// TIA Portal V16 export
// export: Created 2021-11-12T13:31:44.2909433Z, ExportSetting WithDefaults, DisplayName Totally Integrated Automation Portal, DisplayVersion V16 Update 3, DisplayName TIA Portal Version Control Interface, DisplayVersion V16 Update 2, DisplayName TIA Portal Openness, DisplayVersion V16 Update 3, DisplayName SINAMICS Startdrive Advanced, DisplayVersion V16 Update 5, DisplayName SINAMICS Startdrive G130, G150, S120, S150, SINAMICS MV, S210, DisplayVersion V16 Update 5, DisplayName SINAMICS Startdrive G110M, G120, G120C, G120D, G120P, G115D, DisplayVersion V16 Update 5, DisplayName STEP 7 Professional, DisplayVersion V16 Update 3, DisplayName STEP 7 Safety, DisplayVersion V16, DisplayName WinCC UA Professional, DisplayVersion V16 Update 3
FUNCTION_BLOCK "STD_Siemens_MC_Encoder"   // FB31, LAD
TITLE = Siemens MC-Encoder Multiturn 27-bit
{ S7_Optimized_Access := 'TRUE' }
VERSION : 0.1
// MICE standard block 
// Communication with Siemens MC-Encoder Multiturn 27-bit (6FX2001-5FN25)
// 
// 
// Version              Created                        by             Comment
// 0.1                      16.7.2019                   JKu          initial version
// stored: AutoNumber true, IsIECCheckEnabled false, IsRetainMemResEnabled false, MemoryReserve 100, SetENOAutomatically false, UDAEnableTagReadback false
   VAR_INPUT
      IW_HWID : HW_SUBMODULE;
      IB1Preset : Bool;   // Set previously configured home position (absolute)
      IB1Ack : Bool;   // Alarm reset
      IB1AlarmSuppress : Bool;   // Alarm suppression
   END_VAR
   VAR_OUTPUT
      OS_Status : Struct
         Main : "UDT_Status_main";
         Specific : "UDT_MCEncoder_Status_specific";
         Error : "UDT_Error01";
      END_STRUCT;
      OR_AbsPosUnits : Real;   // Absolute actual position [mm]
   END_VAR
   VAR_IN_OUT
      XS_Parameter : "UDT_MCEnkoder_Parameter";   // Individual parameter structure
      XS_Command : "UDT_MCEnkoder_Command";
   END_VAR
   VAR
      SS_Alarm : Struct   // Device alarms
         SensorError : Bool;   // Error in the processing of the sensor signal
         CommandNotSupported : Bool;   // Optional command (in G1_STW) not supported.
         PLCSignOfLifeFailure : Bool;   // The number of permissible failures of the masters
         SynchronizationFault : Bool;   // The number of permissible failures for the bus cycle
         Overflow : Bool;   // The position value in G1_XIST1 overflow
         InvalidData : Bool;   // Data from encoder is invalid and encoder does not respond to commands
         res0_6 : Bool;
         res0_7 : Bool;
      END_STRUCT;
      SS_Warning : Struct   // Device warnings
         res0_0 : Bool;
         res0_1 : Bool;
         res0_2 : Bool;
         res0_3 : Bool;
         res0_4 : Bool;
         res0_5 : Bool;
         res0_6 : Bool;
         res0_7 : Bool;
      END_STRUCT;
   END_VAR
   VAR_TEMP
      TS_Parameter : "UDT_MCEnkoder_Parameter";
      TS_Status : Struct
         Main : "UDT_Status_main";
         Specific : "UDT_MCEncoder_Status_specific";
         Error : "UDT_Error01";
      END_STRUCT;
      TS_InData : "UDT_MCEncoder_I_81";
      TS_OutData : "UDT_MCEncoder_O_81";
      TI_RetVal : Int;
      TI_AbsPosVal : Int;   // Absolute actual position value within one turn
      TR_AbsPosUnits : Real;   // Absolute actual position [mm]
      TI_NoOfRevolution : Int;   // Number of revolutions
      TDWMaskedVal : DWord;   // G1_XIST value masked
      TI_ErrorCode : Int;
      TB1DataValid : Bool;   // Data in G1_XIST1 and G1_ZSW is valid
      TB1 : Bool;
   END_VAR
   VAR CONSTANT
      CI_PulsePerTurn : Int := 8192;   // Resolution
      CI_MaxRevolutions : Int := 16384;   // Maximum number of revolution what the encoder is capable to count
      CI_AbsPosNrOfBits : Int := 13;   // Bit lenght of absolute position value
      CDWMaskAbsPos : DWord := 16#00001FFF;   // Absolute position value mask G1_XIST1
      CDWMaskMultiturnData : DWord := 16#07FFE000;   // Multiturn data mask G1_XIST1
      CDWMaskErrorCode : DWord := 16#00000FFF;   // Error code mask G1_XIST1
   END_VAR
BEGIN

REGION Network 1: Clear temporary variables
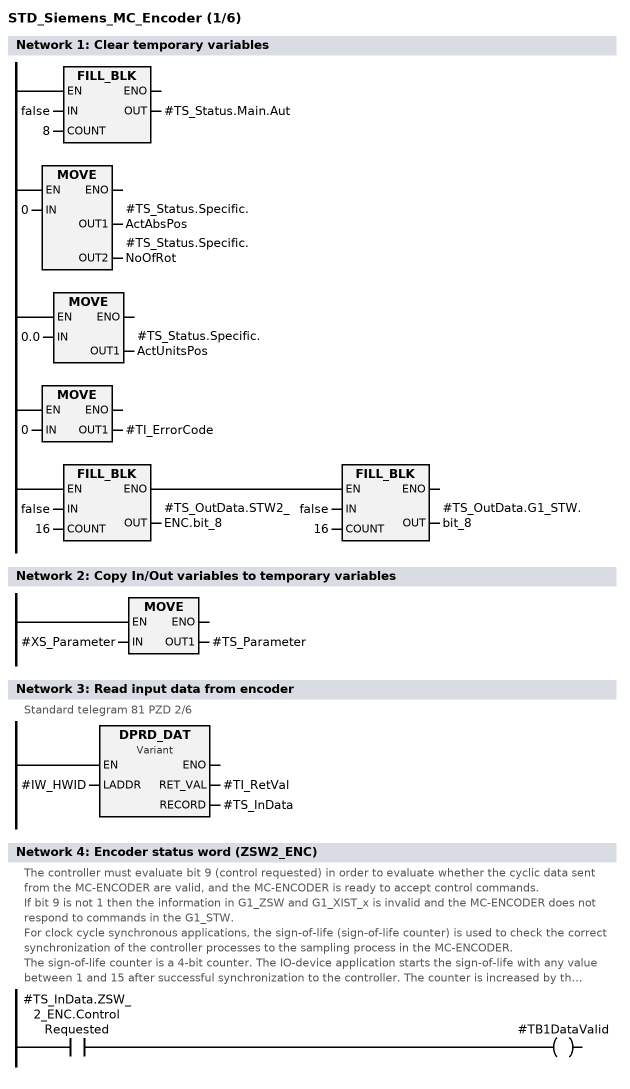
   RUNG wire#powerrail
      FillBlockI(in := false, count := 8, out => #TS_Status.Main.Aut)
   END_RUNG
   RUNG wire#powerrail
      Move(in := 0, out1 => #TS_Status.Specific.ActAbsPos, out2 => #TS_Status.Specific.NoOfRot)
   END_RUNG
   RUNG wire#powerrail
      Move(in := 0.0, out1 => #TS_Status.Specific.ActUnitsPos)
   END_RUNG
   RUNG wire#powerrail
      Move(in := 0, out1 => #TI_ErrorCode)
   END_RUNG
   RUNG wire#powerrail
      FillBlockI(in := false, count := 16, out => #TS_OutData.STW2_ENC.bit_8)
      FillBlockI(in := false, count := 16, out => #TS_OutData.G1_STW.bit_8)
   END_RUNG
   // the same network as SCL:
   FILL_BLK(IN := false, COUNT := 8, OUT => #TS_Status.Main.Aut);
   #TS_Status.Specific.ActAbsPos := 0;
   #TS_Status.Specific.NoOfRot := 0;
   #TS_Status.Specific.ActUnitsPos := 0.0;
   #TI_ErrorCode := 0;
   FILL_BLK(IN := false, COUNT := 16, OUT => #TS_OutData.STW2_ENC.bit_8);
   FILL_BLK(IN := false, COUNT := 16, OUT => #TS_OutData.G1_STW.bit_8);
END_REGION

REGION Network 2: Copy In/Out variables to temporary variables
   RUNG wire#powerrail
      { S7_GenerateENO := "TRUE" } Move(in := #XS_Parameter, out1 => #TS_Parameter)
   END_RUNG
   // the same network as SCL:
   #TS_Parameter := #XS_Parameter;
END_REGION

REGION Network 3: Read input data from encoder
   // Standard telegram 81 PZD 2/6
   RUNG wire#powerrail
      { S7_Templates := "[ptr_type := Variant, laddr_type := HW_IO]" } DPRD_DAT(LADDR := #IW_HWID, RET_VAL => #TI_RetVal, RECORD => #TS_InData)
   END_RUNG
   // the same network as SCL:
   #TI_RetVal := DPRD_DAT(LADDR := #IW_HWID, RECORD => #TS_InData);
END_REGION

REGION Network 4: Encoder status word (ZSW2_ENC)
   // The controller must evaluate bit 9 (control requested) in order to evaluate whether the cyclic data sent from the MC-ENCODER are valid, and the MC-ENCODER is ready to accept control commands.
   // If bit 9 is not 1 then the information in G1_ZSW and G1_XIST_x is invalid and the MC-ENCODER does not respond to commands in the G1_STW.
   // 
   // For clock cycle synchronous applications, the sign-of-life (sign-of-life counter) is used to check the correct synchronization of the controller processes to the sampling process in the MC-ENCODER.
   // The sign-of-life counter is a 4-bit counter. The IO-device application starts the sign-of-life with any value between 1 and 15 after successful synchronization to the controller. The counter is increased by the IO-device in every data cycle. Valid values for the IO-device sign-of-life are 1 to 15, "0" indicates an error and is left out in normal operation.
   // 
   // If the MC-ENCODER identifies an error in the controller sign-of-life, then it stops sending the sign-of-life to the controller. This means that a missing sign-of-life (=0) from the MC-ENCODER to the controller can also be the consequence of an error in the controller sign-of-life to MCENCODER.
   RUNG wire#powerrail
      Contact( #TS_InData.ZSW_2_ENC.ControlRequested )
      Coil( #TB1DataValid )
   END_RUNG
   // the same network as SCL:
   #TB1DataValid := #TS_InData.ZSW_2_ENC.ControlRequested;
END_REGION

REGION Network 5: Sensor status word (G1_ZSW)
   // Signal G1_ZSW is used to control the state machine of the PROFIdrive encoder channel and is the counterpart to control word G1_STW.
   // 
   // bit 11 - Acknowledgement sensor error in process - Is set while requested error acknowledge is processed. Handshake signal related to G1_STW bit 15.
   // bit 12 - Set preset / shift reference point executed - Acknowledgement for "set preset / request shift".
   // bit 13 - Transmit absolute value cyclically - Acknowledgement for "request absolute value cyclically".
   // bit 14 - Parking sensor activated - Acknowledgement for "activate parking sensor". The encoder transmits no valid position value, sensor errors are reset.
   // bit 15 - Sensor error - Indicates a sensor error. A device specific error code is transmitted in G1_XIST2.
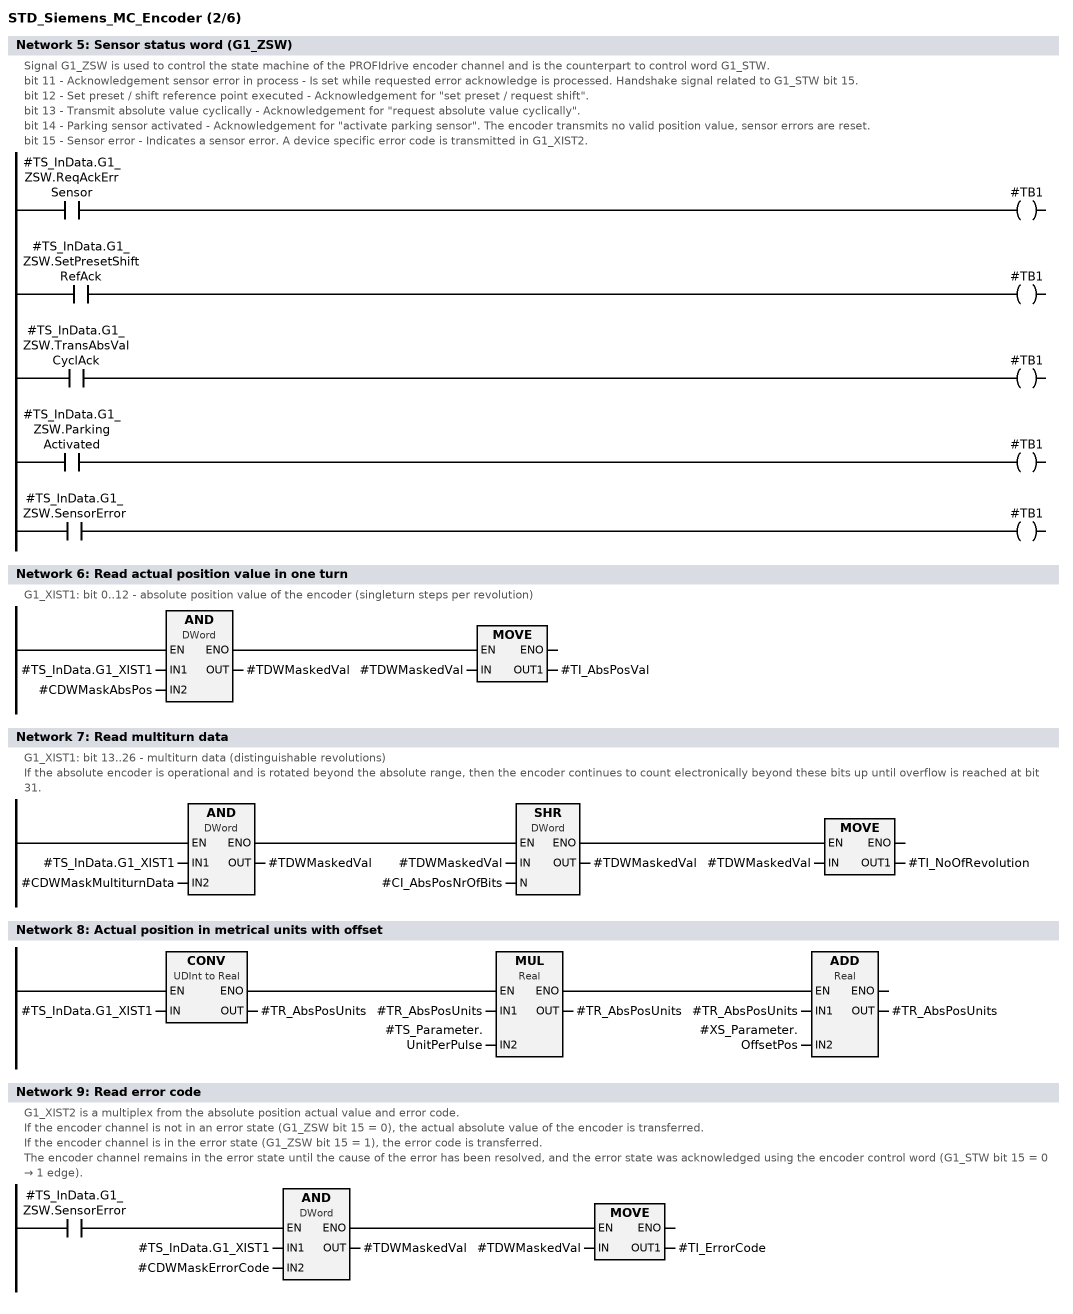
   RUNG wire#powerrail
      Contact( #TS_InData.G1_ZSW.ReqAckErrSensor )
      Coil( #TB1 )
   END_RUNG
   RUNG wire#powerrail
      Contact( #TS_InData.G1_ZSW.SetPresetShiftRefAck )
      Coil( #TB1 )
   END_RUNG
   RUNG wire#powerrail
      Contact( #TS_InData.G1_ZSW.TransAbsValCyclAck )
      Coil( #TB1 )
   END_RUNG
   RUNG wire#powerrail
      Contact( #TS_InData.G1_ZSW.ParkingActivated )
      Coil( #TB1 )
   END_RUNG
   RUNG wire#powerrail
      Contact( #TS_InData.G1_ZSW.SensorError )
      Coil( #TB1 )
   END_RUNG
   // the same network as SCL:
   #TB1 := #TS_InData.G1_ZSW.ReqAckErrSensor;
   #TB1 := #TS_InData.G1_ZSW.SetPresetShiftRefAck;
   #TB1 := #TS_InData.G1_ZSW.TransAbsValCyclAck;
   #TB1 := #TS_InData.G1_ZSW.ParkingActivated;
   #TB1 := #TS_InData.G1_ZSW.SensorError;
END_REGION

REGION Network 6: Read actual position value in one turn
   // G1_XIST1: bit 0..12 - absolute position value of the encoder (singleturn steps per revolution)
   RUNG wire#powerrail
      { S7_Templates := "SrcType := DWord" } And(in1 := #TS_InData.G1_XIST1, in2 := #CDWMaskAbsPos, out => #TDWMaskedVal)
      Move(in := #TDWMaskedVal, out1 => #TI_AbsPosVal)
   END_RUNG
   // the same network as SCL:
   #TDWMaskedVal := #TS_InData.G1_XIST1 AND #CDWMaskAbsPos;
   #TI_AbsPosVal := #TDWMaskedVal;
END_REGION

REGION Network 7: Read multiturn data
   // G1_XIST1: bit 13..26 - multiturn data (distinguishable revolutions)
   // If the absolute encoder is operational and is rotated beyond the absolute range, then the encoder continues to count electronically beyond these bits up until overflow is reached at bit 31.
   RUNG wire#powerrail
      { S7_Templates := "SrcType := DWord" } And(in1 := #TS_InData.G1_XIST1, in2 := #CDWMaskMultiturnData, out => #TDWMaskedVal)
      { S7_Templates := "SrcType := DWord" } Shr(in := #TDWMaskedVal, n := #CI_AbsPosNrOfBits, out => #TDWMaskedVal)
      Move(in := #TDWMaskedVal, out1 => #TI_NoOfRevolution)
   END_RUNG
   // the same network as SCL:
   #TDWMaskedVal := #TS_InData.G1_XIST1 AND #CDWMaskMultiturnData;
   #TDWMaskedVal := SHR(IN := #TDWMaskedVal, N := #CI_AbsPosNrOfBits);
   #TI_NoOfRevolution := #TDWMaskedVal;
END_REGION

REGION Network 8: Actual position in metrical units with offset
   RUNG wire#powerrail
      { S7_Templates := "[SrcType := UDInt, DestType := Real]" } Convert(in := #TS_InData.G1_XIST1, out => #TR_AbsPosUnits)
      { S7_Templates := "SrcType := Real" } Mul(in1 := #TR_AbsPosUnits, in2 := #TS_Parameter.UnitPerPulse, out => #TR_AbsPosUnits)
      { S7_Templates := "SrcType := Real" } Add(in1 := #TR_AbsPosUnits, in2 := #XS_Parameter.OffsetPos, out => #TR_AbsPosUnits)
   END_RUNG
   // the same network as SCL:
   #TR_AbsPosUnits := UDINT_TO_REAL(#TS_InData.G1_XIST1);
   #TR_AbsPosUnits := #TR_AbsPosUnits * #TS_Parameter.UnitPerPulse;
   #TR_AbsPosUnits := #TR_AbsPosUnits + #XS_Parameter.OffsetPos;
END_REGION

REGION Network 9: Read error code
   // G1_XIST2 is a multiplex from the absolute position actual value and error code. 
   // If the encoder channel is not in an error state (G1_ZSW bit 15 = 0), the actual absolute value of the encoder is transferred.
   // If the encoder channel is in the error state (G1_ZSW bit 15 = 1), the error code is transferred.
   // The encoder channel remains in the error state until the cause of the error has been resolved, and the error state was acknowledged using the encoder control word (G1_STW bit 15 = 0 → 1 edge).
   RUNG wire#powerrail
      Contact( #TS_InData.G1_ZSW.SensorError )
      { S7_Templates := "SrcType := DWord" } And(in1 := #TS_InData.G1_XIST1, in2 := #CDWMaskErrorCode, out => #TDWMaskedVal)
      Move(in := #TDWMaskedVal, out1 => #TI_ErrorCode)
   END_RUNG
   // the same network as SCL:
   IF #TS_InData.G1_ZSW.SensorError THEN
       #TDWMaskedVal := #TS_InData.G1_XIST1 AND #CDWMaskErrorCode;
       #TI_ErrorCode := #TDWMaskedVal;
   END_IF;
END_REGION

REGION Network 10: Error evaluation
   // 0x001  Sensor group error - Error in the processing of the sensor signal which causes an invalid Gx_XIST (e.g. electronic malfunction or invalid sensor signal).
   // 0xF01  Command not supported - Optional command (in G1_STW) not supported.
   // 0xF02  Controller sign-of-life failure - The number of permissible failures of the masters sign-of-life was exceeded.
   // 0xF04  Synchronization fault - The number of permissible failures for the bus cycle sign signal was exceeded.
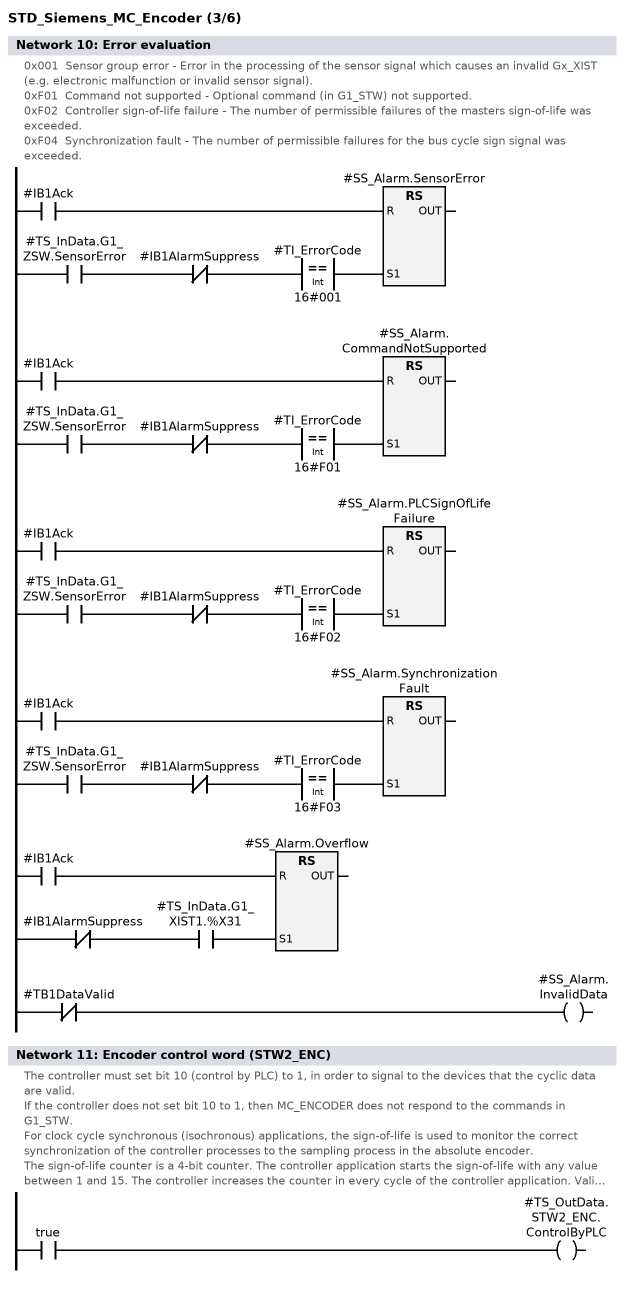
   RUNG wire#powerrail
      Contact( #IB1Ack )
      S_RS(operand := #SS_Alarm.SensorError, s1 := wire#w1)
   END_RUNG
   RUNG wire#powerrail
      Contact( #TS_InData.G1_ZSW.SensorError )
      I_Contact( #IB1AlarmSuppress )
      { S7_Templates := "SrcType := Int" } EQ_Contact(in1 := #TI_ErrorCode, in2 := 16#001)
   END_RUNG wire#w1
   RUNG wire#powerrail
      Contact( #IB1Ack )
      S_RS(operand := #SS_Alarm.CommandNotSupported, s1 := wire#w2)
   END_RUNG
   RUNG wire#powerrail
      Contact( #TS_InData.G1_ZSW.SensorError )
      I_Contact( #IB1AlarmSuppress )
      { S7_Templates := "SrcType := Int" } EQ_Contact(in1 := #TI_ErrorCode, in2 := 16#F01)
   END_RUNG wire#w2
   RUNG wire#powerrail
      Contact( #IB1Ack )
      S_RS(operand := #SS_Alarm.PLCSignOfLifeFailure, s1 := wire#w3)
   END_RUNG
   RUNG wire#powerrail
      Contact( #TS_InData.G1_ZSW.SensorError )
      I_Contact( #IB1AlarmSuppress )
      { S7_Templates := "SrcType := Int" } EQ_Contact(in1 := #TI_ErrorCode, in2 := 16#F02)
   END_RUNG wire#w3
   RUNG wire#powerrail
      Contact( #IB1Ack )
      S_RS(operand := #SS_Alarm.SynchronizationFault, s1 := wire#w4)
   END_RUNG
   RUNG wire#powerrail
      Contact( #TS_InData.G1_ZSW.SensorError )
      I_Contact( #IB1AlarmSuppress )
      { S7_Templates := "SrcType := Int" } EQ_Contact(in1 := #TI_ErrorCode, in2 := 16#F03)
   END_RUNG wire#w4
   RUNG wire#powerrail
      Contact( #IB1Ack )
      S_RS(operand := #SS_Alarm.Overflow, s1 := wire#w5)
   END_RUNG
   RUNG wire#powerrail
      I_Contact( #IB1AlarmSuppress )
      Contact( #TS_InData.G1_XIST1.%X31 )
   END_RUNG wire#w5
   RUNG wire#powerrail
      I_Contact( #TB1DataValid )
      Coil( #SS_Alarm.InvalidData )
   END_RUNG
   // the same network as SCL:
   IF #IB1Ack THEN
       #SS_Alarm.SensorError := FALSE;   // RS flip-flop
   END_IF;
   IF #TS_InData.G1_ZSW.SensorError AND NOT #IB1AlarmSuppress AND (#TI_ErrorCode = 16#001) THEN
       #SS_Alarm.SensorError := TRUE;
   END_IF;
   IF #IB1Ack THEN
       #SS_Alarm.CommandNotSupported := FALSE;   // RS flip-flop
   END_IF;
   IF #TS_InData.G1_ZSW.SensorError AND NOT #IB1AlarmSuppress AND (#TI_ErrorCode = 16#F01) THEN
       #SS_Alarm.CommandNotSupported := TRUE;
   END_IF;
   IF #IB1Ack THEN
       #SS_Alarm.PLCSignOfLifeFailure := FALSE;   // RS flip-flop
   END_IF;
   IF #TS_InData.G1_ZSW.SensorError AND NOT #IB1AlarmSuppress AND (#TI_ErrorCode = 16#F02) THEN
       #SS_Alarm.PLCSignOfLifeFailure := TRUE;
   END_IF;
   IF #IB1Ack THEN
       #SS_Alarm.SynchronizationFault := FALSE;   // RS flip-flop
   END_IF;
   IF #TS_InData.G1_ZSW.SensorError AND NOT #IB1AlarmSuppress AND (#TI_ErrorCode = 16#F03) THEN
       #SS_Alarm.SynchronizationFault := TRUE;
   END_IF;
   IF #IB1Ack THEN
       #SS_Alarm.Overflow := FALSE;   // RS flip-flop
   END_IF;
   IF NOT #IB1AlarmSuppress AND #TS_InData.G1_XIST1.%X31 THEN #SS_Alarm.Overflow := TRUE; END_IF;
   #SS_Alarm.InvalidData := NOT #TB1DataValid;
END_REGION

REGION Network 11: Encoder control word (STW2_ENC)
   // The controller must set bit 10 (control by PLC) to 1, in order to signal to the devices that the cyclic data are valid.
   // If the controller does not set bit 10 to 1, then MC_ENCODER does not respond to the commands in G1_STW.
   // 
   // For clock cycle synchronous (isochronous) applications, the sign-of-life is used to monitor the correct synchronization of the controller processes to the sampling process in the absolute encoder.
   // The sign-of-life counter is a 4-bit counter. The controller application starts the sign-of-life with any value between 1 and 15. The controller increases the counter in every cycle of the controller application. Valid values for the controller sign-of-life are 1 to 15, "0" indicates an error and is left out in normal operation.
   RUNG wire#powerrail
      Contact( true )
      Coil( #TS_OutData.STW2_ENC.ControlByPLC )
   END_RUNG
   // the same network as SCL:
   #TS_OutData.STW2_ENC.ControlByPLC := true;
END_REGION

REGION Network 12: Sensor control word (G1_STW)
   // Signal G1_STW is used to control the state machine of the PROFIdrive encoder channel.
   // 
   // bit 11 - Home position mode - Specifies if the position value shall be set to a previously configured absolute value or shifted by this value. 
   //   0: set home position / preset (absolute) 
   //   1: shift home position / preset (relative = offset)
   // 
   // bit 12 - Set preset / request shift - Preset (resp. shift) is set when changing this bit to "1" (rising edge). Default preset value (shift): 0
   // Note: It can also be parameterized that with a rising edge, the value XIST1 also makes a step.
   // 
   // bit 13 - Request absolute value cyclically - Request of additional cyclic transmission of the absolute actual position in G1_XIST2. If no other data needs to be transferred due to commands or errors the absolute position value will be transmitted automatically.
   // 
   // bit 14 - Activate parking sensor - The encoder is switched inactive and error will be reset. While the encoder is in the parking state, no errors will be generated.
   // 
   // bit 15 - Acknowledging a sensor error - Request to acknowledge / reset a sensor error.
   // 
   // By appropriately parameterizing the absolute encoder, when accepting the preset value, you can set whether this is also directly accepted in G1_XIST1 or G1_XIST3. When the preset value is accepted, this value is also retentively saved automatically. This is to ensure that an absolute value set using preset is also kept after a reset/power up of the encoder.
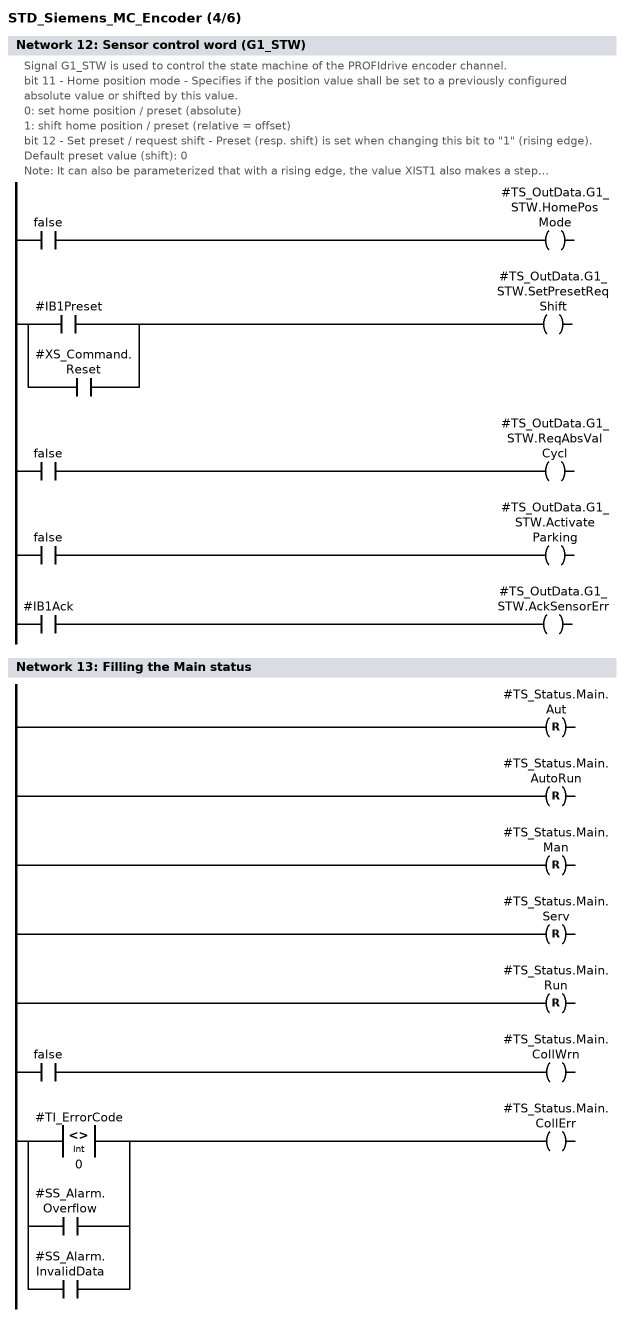
   RUNG wire#powerrail
      Contact( false )
      Coil( #TS_OutData.G1_STW.HomePosMode )
   END_RUNG
   RUNG wire#powerrail
      Contact( #IB1Preset )
      wire#w1
      Coil( #TS_OutData.G1_STW.SetPresetReqShift )
   END_RUNG
   RUNG wire#powerrail
      Contact( #XS_Command.Reset )
   END_RUNG wire#w1
   RUNG wire#powerrail
      Contact( false )
      Coil( #TS_OutData.G1_STW.ReqAbsValCycl )
   END_RUNG
   RUNG wire#powerrail
      Contact( false )
      Coil( #TS_OutData.G1_STW.ActivateParking )
   END_RUNG
   RUNG wire#powerrail
      Contact( #IB1Ack )
      Coil( #TS_OutData.G1_STW.AckSensorErr )
   END_RUNG
   // the same network as SCL:
   #TS_OutData.G1_STW.HomePosMode := false;
   #TS_OutData.G1_STW.SetPresetReqShift := #IB1Preset OR #XS_Command.Reset;
   #TS_OutData.G1_STW.ReqAbsValCycl := false;
   #TS_OutData.G1_STW.ActivateParking := false;
   #TS_OutData.G1_STW.AckSensorErr := #IB1Ack;
END_REGION

REGION Network 13: Filling the Main status
   RUNG wire#powerrail
      R_Coil( #TS_Status.Main.Aut )
   END_RUNG
   RUNG wire#powerrail
      R_Coil( #TS_Status.Main.AutoRun )
   END_RUNG
   RUNG wire#powerrail
      R_Coil( #TS_Status.Main.Man )
   END_RUNG
   RUNG wire#powerrail
      R_Coil( #TS_Status.Main.Serv )
   END_RUNG
   RUNG wire#powerrail
      R_Coil( #TS_Status.Main.Run )
   END_RUNG
   RUNG wire#powerrail
      Contact( false )
      Coil( #TS_Status.Main.CollWrn )
   END_RUNG
   RUNG wire#powerrail
      { S7_Templates := "SrcType := Int" } NE_Contact(in1 := #TI_ErrorCode, in2 := 0)
      wire#w1
      Coil( #TS_Status.Main.CollErr )
   END_RUNG
   RUNG wire#powerrail
      Contact( #SS_Alarm.Overflow )
   END_RUNG wire#w1
   RUNG wire#powerrail
      Contact( #SS_Alarm.InvalidData )
   END_RUNG wire#w1
   // the same network as SCL:
   #TS_Status.Main.Aut := FALSE;
   #TS_Status.Main.AutoRun := FALSE;
   #TS_Status.Main.Man := FALSE;
   #TS_Status.Main.Serv := FALSE;
   #TS_Status.Main.Run := FALSE;
   #TS_Status.Main.CollWrn := false;
   #TS_Status.Main.CollErr := (#TI_ErrorCode <> 0) OR #SS_Alarm.Overflow OR #SS_Alarm.InvalidData;
END_REGION

REGION Network 14: Filling the specific status
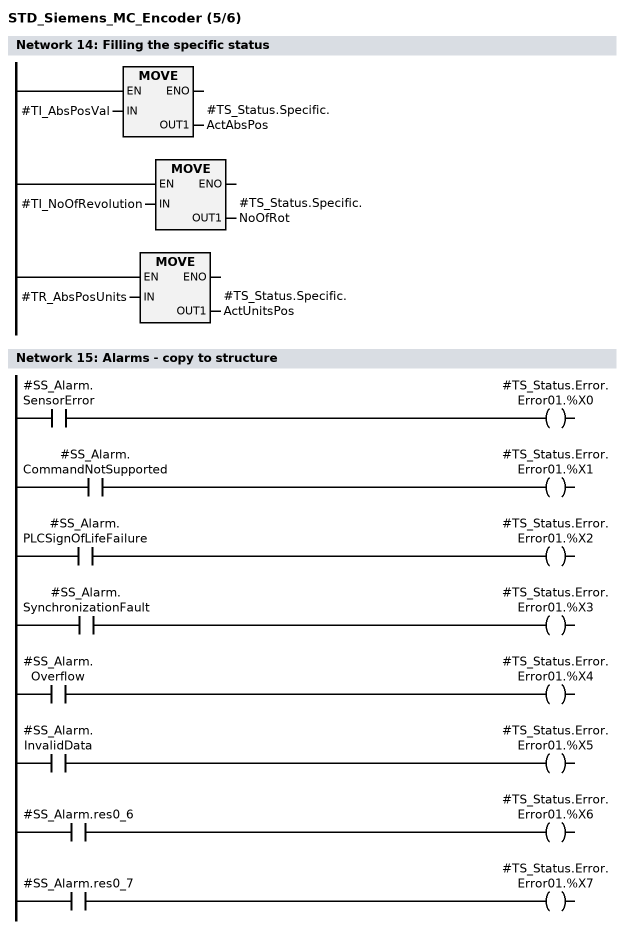
   RUNG wire#powerrail
      Move(in := #TI_AbsPosVal, out1 => #TS_Status.Specific.ActAbsPos)
   END_RUNG
   RUNG wire#powerrail
      Move(in := #TI_NoOfRevolution, out1 => #TS_Status.Specific.NoOfRot)
   END_RUNG
   RUNG wire#powerrail
      Move(in := #TR_AbsPosUnits, out1 => #TS_Status.Specific.ActUnitsPos)
   END_RUNG
   // the same network as SCL:
   #TS_Status.Specific.ActAbsPos := #TI_AbsPosVal;
   #TS_Status.Specific.NoOfRot := #TI_NoOfRevolution;
   #TS_Status.Specific.ActUnitsPos := #TR_AbsPosUnits;
END_REGION

REGION Network 15: Alarms - copy to structure
   RUNG wire#powerrail
      Contact( #SS_Alarm.SensorError )
      Coil( #TS_Status.Error.Error01.%X0 )
   END_RUNG
   RUNG wire#powerrail
      Contact( #SS_Alarm.CommandNotSupported )
      Coil( #TS_Status.Error.Error01.%X1 )
   END_RUNG
   RUNG wire#powerrail
      Contact( #SS_Alarm.PLCSignOfLifeFailure )
      Coil( #TS_Status.Error.Error01.%X2 )
   END_RUNG
   RUNG wire#powerrail
      Contact( #SS_Alarm.SynchronizationFault )
      Coil( #TS_Status.Error.Error01.%X3 )
   END_RUNG
   RUNG wire#powerrail
      Contact( #SS_Alarm.Overflow )
      Coil( #TS_Status.Error.Error01.%X4 )
   END_RUNG
   RUNG wire#powerrail
      Contact( #SS_Alarm.InvalidData )
      Coil( #TS_Status.Error.Error01.%X5 )
   END_RUNG
   RUNG wire#powerrail
      Contact( #SS_Alarm.res0_6 )
      Coil( #TS_Status.Error.Error01.%X6 )
   END_RUNG
   RUNG wire#powerrail
      Contact( #SS_Alarm.res0_7 )
      Coil( #TS_Status.Error.Error01.%X7 )
   END_RUNG
   // the same network as SCL:
   #TS_Status.Error.Error01.%X0 := #SS_Alarm.SensorError;
   #TS_Status.Error.Error01.%X1 := #SS_Alarm.CommandNotSupported;
   #TS_Status.Error.Error01.%X2 := #SS_Alarm.PLCSignOfLifeFailure;
   #TS_Status.Error.Error01.%X3 := #SS_Alarm.SynchronizationFault;
   #TS_Status.Error.Error01.%X4 := #SS_Alarm.Overflow;
   #TS_Status.Error.Error01.%X5 := #SS_Alarm.InvalidData;
   #TS_Status.Error.Error01.%X6 := #SS_Alarm.res0_6;
   #TS_Status.Error.Error01.%X7 := #SS_Alarm.res0_7;
END_REGION

REGION Network 16: Warnings - copy to structure
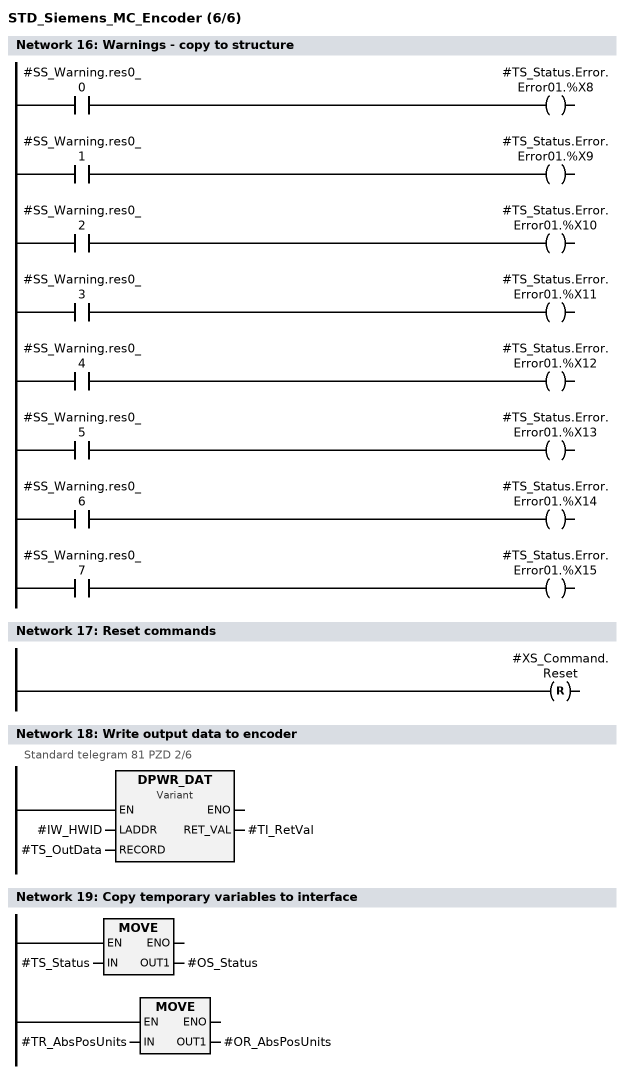
   RUNG wire#powerrail
      Contact( #SS_Warning.res0_0 )
      Coil( #TS_Status.Error.Error01.%X8 )
   END_RUNG
   RUNG wire#powerrail
      Contact( #SS_Warning.res0_1 )
      Coil( #TS_Status.Error.Error01.%X9 )
   END_RUNG
   RUNG wire#powerrail
      Contact( #SS_Warning.res0_2 )
      Coil( #TS_Status.Error.Error01.%X10 )
   END_RUNG
   RUNG wire#powerrail
      Contact( #SS_Warning.res0_3 )
      Coil( #TS_Status.Error.Error01.%X11 )
   END_RUNG
   RUNG wire#powerrail
      Contact( #SS_Warning.res0_4 )
      Coil( #TS_Status.Error.Error01.%X12 )
   END_RUNG
   RUNG wire#powerrail
      Contact( #SS_Warning.res0_5 )
      Coil( #TS_Status.Error.Error01.%X13 )
   END_RUNG
   RUNG wire#powerrail
      Contact( #SS_Warning.res0_6 )
      Coil( #TS_Status.Error.Error01.%X14 )
   END_RUNG
   RUNG wire#powerrail
      Contact( #SS_Warning.res0_7 )
      Coil( #TS_Status.Error.Error01.%X15 )
   END_RUNG
   // the same network as SCL:
   #TS_Status.Error.Error01.%X8 := #SS_Warning.res0_0;
   #TS_Status.Error.Error01.%X9 := #SS_Warning.res0_1;
   #TS_Status.Error.Error01.%X10 := #SS_Warning.res0_2;
   #TS_Status.Error.Error01.%X11 := #SS_Warning.res0_3;
   #TS_Status.Error.Error01.%X12 := #SS_Warning.res0_4;
   #TS_Status.Error.Error01.%X13 := #SS_Warning.res0_5;
   #TS_Status.Error.Error01.%X14 := #SS_Warning.res0_6;
   #TS_Status.Error.Error01.%X15 := #SS_Warning.res0_7;
END_REGION

REGION Network 17: Reset commands
   RUNG wire#powerrail
      R_Coil( #XS_Command.Reset )
   END_RUNG
   // the same network as SCL:
   #XS_Command.Reset := FALSE;
END_REGION

REGION Network 18: Write output data to encoder
   // Standard telegram 81 PZD 2/6
   RUNG wire#powerrail
      { S7_Templates := "[ptr_type := Variant, laddr_type := HW_IO]" } DPWR_DAT(LADDR := #IW_HWID, RECORD := #TS_OutData, RET_VAL => #TI_RetVal)
   END_RUNG
   // the same network as SCL:
   #TI_RetVal := DPWR_DAT(LADDR := #IW_HWID, RECORD := #TS_OutData);
END_REGION

REGION Network 19: Copy temporary variables to interface
   RUNG wire#powerrail
      { S7_GenerateENO := "TRUE" } Move(in := #TS_Status, out1 => #OS_Status)
   END_RUNG
   RUNG wire#powerrail
      Move(in := #TR_AbsPosUnits, out1 => #OR_AbsPosUnits)
   END_RUNG
   // the same network as SCL:
   #OS_Status := #TS_Status;
   #OR_AbsPosUnits := #TR_AbsPosUnits;
END_REGION
END_FUNCTION_BLOCK
